(* GVLs/GLOBAL_VARS *)

{attribute 'qualified_only'}
VAR_GLOBAL
    DO_EL2008_0    AT %Q* : BOOL;   // EL2008 channel 1
    DO_EL2008_1    AT %Q* : BOOL;   // EL2008 channel 2

  	// — these must sit on WORD I/O addresses, not bit addresses —  
	PCin  AT %IW0 : PcComInData;   // 66‐byte input image = SerStatus:WORD + D[0..63]
	PCout AT %QW0 : PcComOutData;  // 66‐byte output image = SerCtrl:WORD + D[0..63]  
END_VAR

(* stored: Version 1.1.0.1
   GVL GLOBAL_VARS: Id {a07ed368-aff3-40fe-9fbb-b210d5bb7bb2} *)
